RoboDK station: DemoFactorySimulation.rdk

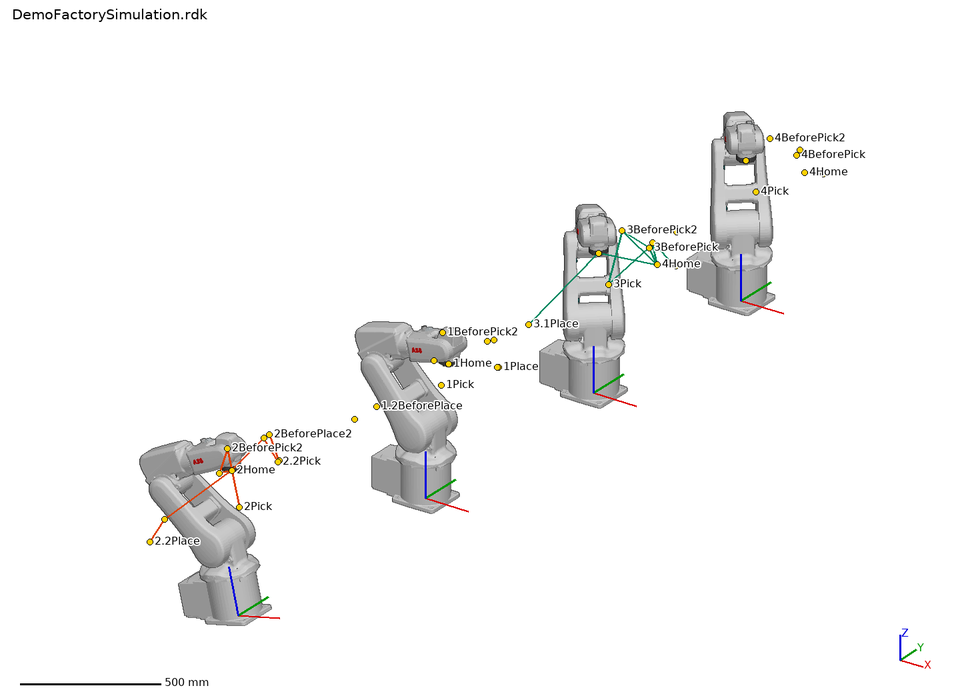
[picture v0: the station drawn from its stored meshes, robots at their saved joint values, targets as dots, program paths as lines]
Station RDTSDemoBasketLine. Poses are relative to the parent item; angles as X-Y-Z fixed-axis rotations.
Station parameters (name, value as stored): 1MoveToPick, 0, 1MakePick, 0, 1PickObjOK, 0, 1MoveToPlace, 0, 1MakePlace, 0, 1PlaceObjOK, 0, 1Waitting, 1, 2MoveToPick, 0, 2MakePick, 0, 2PickObjOK, 1, 2MoveToPlace, 0, 2MakePlace, 0, 2PlaceObjOK, 0, 2Waitting, 1, 3MoveToPick, 0, 3MakePick, 1, 3PickObjOK, 0, 3MoveToPlace, 0, 3MakePlace, 0, 3PlaceObjOK, 0, 3Waitting, 0, 4MoveToPick, 0, 4MakePick, 0, 4PickObjOK, 0, 4MoveToPlace, 0, 4MakePlace, 0, 4PlaceObjOK, 0, 4Waitting, 1, 5MoveToPick, 0, 5MakePick, 0, 5PickObjOK, 0, 5MoveToPlace, 0, 5MakePlace, 0, 5PlaceObjOK, 0, 5Waitting, 1
  - frame Robot1Base at (0, 605.93, 0) mm
    - robot Robot1 (model ABB IRB 120-3/0.6): 6 axes, payload 3 kg, reach 580 mm, repeatability 0.01 mm, weight 25 kg
        modified DH rows (alpha deg, a mm, theta deg, d mm): 0, 0, 0, 290; -90, 0, -90, 0; 0, 270, 0, 0; -90, 70, 0, 302; 90, 0, 0, 0; -90, 0, 180, 72
        joint limits [-165, -110, -90, -160, -120, -400] to [165, 110, 70, 160, 120, 400]; home [0, 0, 0, 0, 0, 0]; saved at [0, -40.936, 28.088, 0, 105.49, 0]
    - target 1Home (Cartesian target) at (98.64, 0, 557.45) mm, rotated rx 180 ry -2.64 rz 180 deg; joints [0, -40.936, 28.088, 0, 105.49, 0] of Robot1
    - target 1BeforePick (Cartesian target) at (1.46, 49.24, 523.75) mm, rotated rx -179.78 ry 0.01 rz -91.44 deg; joints [88.62, -55.08, 38.94, -0.23, 106.13, 0] of Robot1
    - target 1BeforePick2 (Cartesian target) at (-74.07, 211.85, 549) mm, rotated rx -179.78 ry 0 rz -89.11 deg; joints [109.338, -16.563, 16.145, -0.21, 90.487, 18.449] of Robot1
    - target 1Pick (Cartesian target) at (-133.52, 287.77, 294.7) mm, rotated rx -179.78 ry 0.01 rz -90.69 deg; joints [114.936, 14.64, 34.94, -0.312, 40.509, 25.866] of Robot1
    - target 1AfterPick (Cartesian target) at (-74.07, 211.85, 549) mm, rotated rx -179.78 ry 0 rz -89.11 deg; joints [109.338, -16.563, 16.145, -0.21, 90.487, 18.449] of Robot1
    - target 1AfterPick2 (Cartesian target) at (1.46, 49.24, 523.75) mm, rotated rx -179.78 ry 0.01 rz -91.44 deg; joints [88.62, -55.08, 38.94, -0.23, 106.13, 0] of Robot1
    - target 1BeforePlace (Cartesian target) at (237.81, 40.67, 670.65) mm, rotated rx 180 ry -2.64 rz -180 deg; joints [9.575, -1.266, -21.78, 0.487, 115.649, 9.776] of Robot1
    - target 1BeforePlace2 (Cartesian target) at (266.26, 40.67, 684.58) mm, rotated rx 180 ry -2.64 rz 180 deg; joints [8.58, 7.385, -34.207, 0.452, 119.433, 8.793] of Robot1
    - target 1Place (Cartesian target) at (293.03, 32.57, 586.26) mm, rotated rx 180 ry -2.64 rz -180 deg; joints [6.273, 0.868, -6.289, 0.291, 98.045, 6.307] of Robot1
    - target 1AfterPlace (Cartesian target) at (266.26, 40.67, 684.58) mm, rotated rx 180 ry -2.64 rz 180 deg; joints [8.58, 7.385, -34.207, 0.452, 119.433, 8.793] of Robot1
    - target 1AfterPlace2 (Cartesian target) at (237.81, 40.67, 670.65) mm, rotated rx 180 ry -2.64 rz 180 deg; joints [9.575, -1.266, -21.78, 0.487, 115.649, 9.776] of Robot1
    - target 1.2BeforePick (Cartesian target) at (237.81, 40.67, 670.65) mm, rotated rx -180 ry -2.64 rz -180 deg; joints [9.575, -1.266, -21.78, 0.487, 115.649, 9.776] of Robot1
    - target 1.2Pick (Cartesian target) at (287.41, 32.18, 584.86) mm, rotated rx -180 ry -2.64 rz -180 deg; joints [6.316, -0.426, -4.718, 0.293, 97.768, 6.349] of Robot1
    - target 1.2AfterPick (Cartesian target) at (237.81, 40.67, 670.65) mm, rotated rx -180 ry -2.64 rz -180 deg; joints [9.575, -1.266, -21.78, 0.487, 115.649, 9.776] of Robot1
    - target 1.2BeforePlace (Cartesian target) at (0, -302, 481.65) mm, rotated rx 180 ry 0 rz 90 deg; joints [-90, -1.686, 15.888, 0, 75.798, 0] of Robot1
    - target 1.2Place (Cartesian target) at (-151.28, -221.68, 357.52) mm, rotated rx 180 ry 0 rz 90 deg; joints [-124.31, -2.755, 40.632, 0, 52.123, -34.31] of Robot1
    - target 1.2AfterPlace (Cartesian target) at (0, -302, 481.65) mm, rotated rx 180 ry 0 rz 90 deg; joints [-90, -1.686, 15.888, 0, 75.798, 0] of Robot1
  - program RobotProg1 (59 instructions, listed below)
  - frame Robot2Base at (0, -551.31, 0) mm, rotated rx 0 ry -12.89 rz 0 deg
    - robot Robot2 (model ABB IRB 120-3/0.6): 6 axes, payload 3 kg, reach 580 mm, repeatability 0.01 mm, weight 25 kg
        modified DH rows (alpha deg, a mm, theta deg, d mm): 0, 0, 0, 290; -90, 0, -90, 0; 0, 270, 0, 0; -90, 70, 0, 302; 90, 0, 0, 0; -90, 0, 180, 72
        joint limits [-165, -110, -90, -160, -120, -400] to [165, 110, 70, 160, 120, 400]; home [0, 0, 0, 0, 0, 0]; saved at [0, -40.936, 28.088, 0, 105.49, 0]
    - target 2Home (Cartesian target) at (98.64, 0, 557.45) mm, rotated rx 180 ry -2.64 rz 180 deg; joints [0, -40.936, 28.088, 0, 105.49, 0] of Robot2
    - target 2BeforePick (Cartesian target) at (1.46, 49.24, 523.75) mm, rotated rx -179.78 ry 0.01 rz -91.44 deg; joints [88.62, -55.08, 38.94, -0.23, 106.13, 0] of Robot2
    - target 2BeforePick2 (Cartesian target) at (-74.07, 211.85, 549) mm, rotated rx -179.78 ry 0 rz -89.11 deg; joints [109.338, -16.563, 16.145, -0.21, 90.487, 18.449] of Robot2
    - target 2Pick (Cartesian target) at (-133.52, 287.77, 294.7) mm, rotated rx -179.78 ry 0.01 rz -91.91 deg; joints [114.936, 14.64, 34.94, -0.312, 40.509, 27.079] of Robot2
    - target 2AfterPick (Cartesian target) at (-74.07, 211.85, 549) mm, rotated rx -179.78 ry 0 rz -89.11 deg; joints [109.338, -16.563, 16.145, -0.21, 90.487, 18.449] of Robot2
    - target 2AfterPick2 (Cartesian target) at (1.46, 49.24, 523.75) mm, rotated rx -179.78 ry 0.01 rz -91.44 deg; joints [88.62, -55.08, 38.94, -0.23, 106.13, 0] of Robot2
    - target 2BeforePlace (Cartesian target) at (237.81, 40.67, 670.65) mm, rotated rx 180 ry -2.64 rz -180 deg; joints [9.575, -1.266, -21.78, 0.487, 115.649, 9.776] of Robot2
    - target 2BeforePlace2 (Cartesian target) at (266.26, 40.67, 684.58) mm, rotated rx 180 ry -2.64 rz 180 deg; joints [8.58, 7.385, -34.207, 0.452, 119.433, 8.793] of Robot2
    - target 2Place (Cartesian target) at (293.25, 32.57, 591.05) mm, rotated rx 180 ry -2.64 rz 180 deg; joints [6.268, 1.267, -7.631, 0.292, 98.989, 6.307] of Robot2
    - target 2AfterPlace (Cartesian target) at (266.26, 40.67, 684.58) mm, rotated rx 180 ry -2.64 rz 180 deg; joints [8.58, 7.385, -34.207, 0.452, 119.433, 8.793] of Robot2
    - target 2AfterPlace2 (Cartesian target) at (237.81, 40.67, 670.65) mm, rotated rx 180 ry -2.64 rz 180 deg; joints [9.575, -1.266, -21.78, 0.487, 115.649, 9.776] of Robot2
    - target 2.2BeforePick (Cartesian target) at (237.81, 40.67, 670.65) mm, rotated rx -180 ry -2.64 rz -180 deg; joints [9.575, -1.266, -21.78, 0.487, 115.649, 9.776] of Robot2
    - target 2.2Pick (Cartesian target) at (287.41, 32.18, 584.86) mm, rotated rx -180 ry -2.64 rz -180 deg; joints [6.316, -0.426, -4.718, 0.293, 97.768, 6.349] of Robot2
    - target 2.2AfterPick (Cartesian target) at (237.81, 40.67, 670.65) mm, rotated rx -180 ry -2.64 rz -180 deg; joints [9.575, -1.266, -21.78, 0.487, 115.649, 9.776] of Robot2
    - target 2.2BeforePlace (Cartesian target) at (0, -302, 481.65) mm, rotated rx 180 ry 0 rz 90 deg; joints [-90, -1.686, 15.888, 0, 75.798, 0] of Robot2
    - target 2.2Place (Cartesian target) at (-151.28, -221.68, 357.52) mm, rotated rx 180 ry 0 rz 90 deg; joints [-124.31, -2.755, 40.632, 0, 52.123, -34.31] of Robot2
    - target 2.2AfterPlace (Cartesian target) at (0, -302, 481.65) mm, rotated rx 180 ry 0 rz 90 deg; joints [-90, -1.686, 15.888, 0, 75.798, 0] of Robot2
  - program RobotProg2 (59 instructions, listed below)
  - frame Robot3Base at (0, 1644.74, 0) mm
    - robot Robot3 (model ABB IRB 120-3/0.6): 6 axes, payload 3 kg, reach 580 mm, repeatability 0.01 mm, weight 25 kg
        modified DH rows (alpha deg, a mm, theta deg, d mm): 0, 0, 0, 290; -90, 0, -90, 0; 0, 270, 0, 0; -90, 70, 0, 302; 90, 0, 0, 0; -90, 0, 180, 72
        joint limits [-165, -110, -90, -160, -120, -400] to [165, 110, 70, 160, 120, 400]; home [0, 0, 0, 0, 0, 0]; saved at [-48.899, -24.574, 6.021, 0.542, 108.231, 40.826]
    - target 4Home (Cartesian target) at (262.7, 17.2, 573.39) mm, rotated rx 179.91 ry 0.6 rz -179.52 deg; joints [3.731, -7.418, 4.046, 0.057, 92.769, 3.257] of Robot3
    - target 3BeforePick (Cartesian target) at (168.05, 102.25, 580.49) mm, rotated rx 175.96 ry 3.61 rz -144.21 deg; joints [29.71, -21.07, 13.293, 4.417, 94.607, -5.734] of Robot3
    - target 3BeforePick2 (Cartesian target) at (16.7, 152.98, 583.81) mm, rotated rx -179.66 ry 5.4 rz -92.3 deg; joints [83.754, -29.723, 17.773, 0.036, 96.534, -3.924] of Robot3
    - target 3Pick (Cartesian target) at (-130.61, 278.87, 281.48) mm, rotated rx -179.66 ry 5.4 rz -92.3 deg; joints [115.76, 13.813, 39.181, -5.284, 32.502, 32.421] of Robot3
    - target 3Place (Cartesian target) at (339.21, 24.19, 586.4) mm, rotated rx 179.91 ry 0.6 rz -179.52 deg; joints [4.067, 9.967, -16.219, 0.054, 95.647, 3.595] of Robot3
    - target 3BeforePlace (Cartesian target) at (240.47, 19.38, 654.16) mm, rotated rx 179.91 ry 0.6 rz -179.52 deg; joints [4.594, -4.403, -15.131, 0.051, 108.929, 4.134] of Robot3
    - target 3.1Place (Cartesian target) at (-136.77, -205.36, 314.46) mm, rotated rx 179.4 ry -0.09 rz 90.45 deg; joints [-123.793, -2.069, 49.122, 0.647, 43.362, -34.71] of Robot3
    - target 3.1BeforePlace (Cartesian target) at (100.51, -114.23, 626) mm, rotated rx 179.4 ry -0.09 rz 90.45 deg; joints [-48.899, -24.574, 6.021, 0.542, 108.231, 40.826] of Robot3
  - program RobotProg3 (59 instructions, listed below)
  - frame RobotBase4 at (0, 2557.3, 0) mm
    - robot Robot4 (model ABB IRB 120-3/0.6): 6 axes, payload 3 kg, reach 580 mm, repeatability 0.01 mm, weight 25 kg
        modified DH rows (alpha deg, a mm, theta deg, d mm): 0, 0, 0, 290; -90, 0, -90, 0; 0, 270, 0, 0; -90, 70, 0, 302; 90, 0, 0, 0; -90, 0, 180, 72
        joint limits [-165, -110, -90, -160, -120, -400] to [165, 110, 70, 160, 120, 400]; home [0, 0, 0, 0, 0, 0]; saved at [-48.899, -24.574, 6.021, 0.542, 108.231, 40.826]
    - target 4Home (Cartesian target) at (262.7, 17.2, 573.39) mm, rotated rx 179.91 ry 0.6 rz -179.52 deg; joints [3.731, -7.418, 4.046, 0.057, 92.769, 3.257] of Robot4
    - target 4BeforePick (Cartesian target) at (168.05, 102.25, 580.49) mm, rotated rx 175.96 ry 3.61 rz -144.21 deg; joints [29.71, -21.07, 13.293, 4.417, 94.607, -5.734] of Robot4
    - target 4BeforePick2 (Cartesian target) at (16.7, 152.98, 583.81) mm, rotated rx -179.66 ry 5.4 rz -92.3 deg; joints [83.754, -29.723, 17.773, 0.036, 96.534, -3.924] of Robot4
    - target 4Pick (Cartesian target) at (-130.61, 278.87, 281.48) mm, rotated rx -179.66 ry 5.4 rz -92.3 deg; joints [115.76, 13.813, 39.181, -5.284, 32.502, 32.421] of Robot4
    - target 4Place (Cartesian target) at (339.21, 24.19, 586.4) mm, rotated rx 179.91 ry 0.6 rz -179.52 deg; joints [4.067, 9.967, -16.219, 0.054, 95.647, 3.595] of Robot4
    - target 4BeforePlace (Cartesian target) at (240.47, 19.38, 654.16) mm, rotated rx 179.91 ry 0.6 rz -179.52 deg; joints [4.594, -4.403, -15.131, 0.051, 108.929, 4.134] of Robot4
    - target 4.1Place (Cartesian target) at (-136.77, -205.36, 314.46) mm, rotated rx 179.4 ry -0.09 rz 90.45 deg; joints [-123.793, -2.069, 49.122, 0.647, 43.362, -34.71] of Robot4
    - target 4.1BeforePlace (Cartesian target) at (100.51, -114.23, 626) mm, rotated rx 179.4 ry -0.09 rz 90.45 deg; joints [-48.899, -24.574, 6.021, 0.542, 108.231, 40.826] of Robot4
  - program RobotProg3 (59 instructions, listed below)
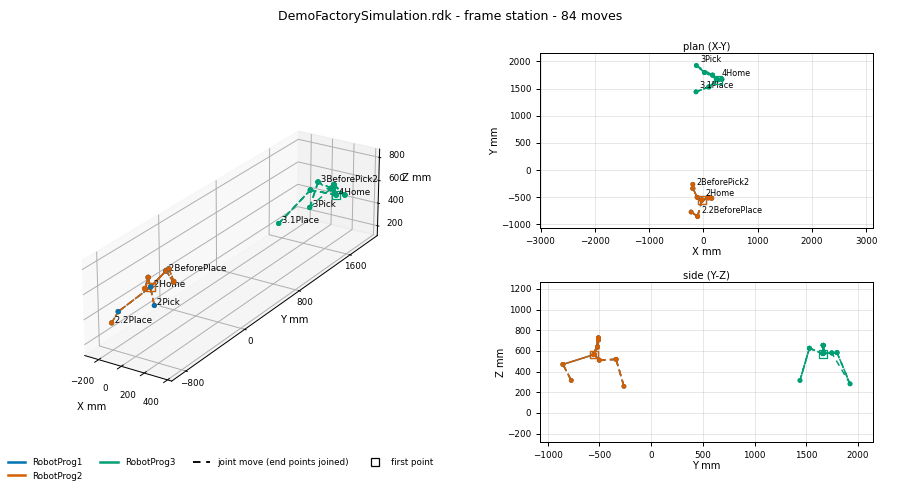
[picture p0: tool path of DemoFactorySimulation.rdk in frame station, 84 of 84 moves have a stored position in this frame; points joined in program order, loops and branches not executed]

--- program RobotProg1 (robot Robot1) ---
  Set Ref.: Robot1Base
  MoveJ (2Home)
  Set 1MakePick=0
  Set 1PickObjOK=0
  Set 1MakePlace=0
  Set 1PlaceObjOK=0
  Wait 1MoveToPick=1
  Set 1Waitting=0
  MoveJ (2BeforePick)
  MoveJ (2BeforePick2)
  MoveJ (2Pick)
  Set 1MakePick=1
  Wait 1PickObjOK=1
  Set 1MakePick=0
  暂停 2.0 s
  MoveJ (2AfterPick)
  MoveJ (2AfterPick2)
  MoveJ (2Home)
  Set 1Waitting=1
  Wait 1MoveToPlace=1
  Set 1Waitting=0
  MoveJ (2BeforePlace)
  MoveJ (2BeforePlace2)
  MoveJ (2Place)
  Set 1MakePlace=1
  Wait 1PlaceObjOK=1
  Set 1MakePlace=0
  暂停 1.0 s
  MoveJ (2AfterPlace)
  MoveJ (2AfterPlace2)
  MoveJ (2Home)
  Set 1Waitting=1
  暂停 2.5 s
  Set 1MakePick=0
  Set 1PickObjOK=0
  Set 1MakePlace=0
  Set 1PlaceObjOK=0
  Wait 1MoveToPick=1
  Set 1Waitting=0
  MoveJ (2.2BeforePick)
  MoveJ (2.2Pick)
  Set 1MakePick=1
  Wait 1PickObjOK=1
  Set 1MakePick=0
  暂停 2.0 s
  MoveJ (2.2AfterPick)
  MoveJ (2Home)
  Set 1Waitting=1
  Wait 1MoveToPlace=1
  Set 1Waitting=0
  MoveJ (2.2BeforePlace)
  MoveJ (2.2Place)
  Set 1MakePlace=1
  Wait 1PlaceObjOK=1
  Set 1MakePlace=0
  暂停 1.0 s
  MoveJ (2.2AfterPlace)
  MoveJ (2Home)
  Set 1Waitting=1

--- program RobotProg2 (robot Robot2) ---
  设置参考: Robot2Base
  MoveJ (2Home)
  Set 2MakePick=0
  Set 2PickObjOK=0
  Set 2MakePlace=0
  Set 2PlaceObjOK=0
  Wait 2MoveToPick=1
  Set 2Waitting=0
  MoveJ (2BeforePick)
  MoveJ (2BeforePick2)
  MoveJ (2Pick)
  Set 2MakePick=1
  Wait 2PickObjOK=1
  Set 2MakePick=0
  暂停 2.0 s
  MoveJ (2AfterPick)
  MoveJ (2AfterPick2)
  MoveJ (2Home)
  Set 2Waitting=1
  Wait 2MoveToPlace=1
  Set 2Waitting=0
  MoveJ (2BeforePlace)
  MoveJ (2BeforePlace2)
  MoveJ (2Place)
  Set 2MakePlace=1
  Wait 2PlaceObjOK=1
  Set 2MakePlace=0
  暂停 1.0 s
  MoveJ (2AfterPlace)
  MoveJ (2AfterPlace2)
  MoveJ (2Home)
  Set 2Waitting=1
  暂停 2.5 s
  Set 2MakePick=0
  Set 2PickObjOK=0
  Set 2MakePlace=0
  Set 2PlaceObjOK=0
  Wait 2MoveToPick=1
  Set 2Waitting=0
  MoveJ (2.2BeforePick)
  MoveJ (2.2Pick)
  Set 2MakePick=1
  Wait 2PickObjOK=1
  Set 2MakePick=0
  暂停 2.0 s
  MoveJ (2.2AfterPick)
  MoveJ (2Home)
  Set 2Waitting=1
  Wait 2MoveToPlace=1
  Set 2Waitting=0
  MoveJ (2.2BeforePlace)
  MoveJ (2.2Place)
  Set 2MakePlace=1
  Wait 2PlaceObjOK=1
  Set 2MakePlace=0
  暂停 1.0 s
  MoveJ (2.2AfterPlace)
  MoveJ (2Home)
  Set 2Waitting=1

--- program RobotProg3 (robot Robot3) ---
  Set Ref.: Robot3Base
  MoveJ (3Home) -> target 4Home
  Set 3MakePick=0
  Set 3PickObjOK=0
  Set 3MakePlace=0
  Set 3PlaceObjOK=0
  Wait 3MoveToPick=1
  Set 3Waitting=0
  MoveJ (3BeforePick)
  MoveJ (3BeforePick2)
  MoveJ (3Pick)
  Set 3MakePick=1
  Wait 3PickObjOK=1
  Set 3MakePick=0
  暂停 2.0 s
  MoveJ (3BeforePick) -> target 3BeforePick2
  MoveJ (3BeforePick) -> target 3BeforePick2
  MoveJ (3Home) -> target 4Home
  Set 3Waitting=1
  Wait 3MoveToPlace=1
  Set 3Waitting=0
  MoveJ (3BeforePlace)
  MoveJ (3BeforePlace)
  MoveJ (3Place)
  Set 3MakePlace=1
  Wait 3PlaceObjOK=1
  Set 3MakePlace=0
  暂停 1.0 s
  MoveJ (3BeforePlace)
  MoveJ (3BeforePlace)
  MoveJ (3Home) -> target 4Home
  Set 3Waitting=1
  暂停 2.5 s
  Set 3MakePick=0
  Set 3PickObjOK=0
  Set 3MakePlace=0
  Set 3PlaceObjOK=0
  Wait 3MoveToPick=1
  Set 3Waitting=0
  MoveJ (3BeforePlace)
  MoveJ (3Place)
  Set 3MakePick=1
  Wait 3PickObjOK=1
  Set 3MakePick=0
  暂停 2.0 s
  MoveJ (3BeforePlace)
  MoveJ (3Home) -> target 4Home
  Set 3Waitting=1
  Wait 3MoveToPlace=1
  Set 3Waitting=0
  MoveJ (3.1BeforePlace)
  MoveJ (3.1Place)
  Set 3MakePlace=1
  Wait 3PlaceObjOK=1
  Set 3MakePlace=0
  暂停 1.0 s
  MoveJ (3.1BeforePlace)
  MoveJ (3Home) -> target 4Home
  Set 3Waitting=1

--- program RobotProg3 (robot Robot4) ---
  Set Ref.: RobotBase4
  MoveJ (4Home)
  Set 4MakePick=0
  Set 4PickObjOK=0
  Set 4MakePlace=0
  Set 4PlaceObjOK=0
  Wait 4MoveToPick=1
  Set 4Waitting=0
  MoveJ (4BeforePick) -> target 3BeforePick
  MoveJ (4BeforePick2) -> target 3BeforePick2
  MoveJ (4Pick) -> target 3Pick
  Set 4MakePick=1
  Wait 4PickObjOK=1
  Set 4MakePick=0
  暂停 2.0 s
  MoveJ (3BeforePick)
  MoveJ (3BeforePick)
  MoveJ (4Home)
  Set 4Waitting=1
  Wait 4MoveToPlace=1
  Set 4Waitting=0
  MoveJ (3BeforePlace)
  MoveJ (3BeforePlace)
  MoveJ (3Place)
  Set 4MakePlace=1
  Wait 4PlaceObjOK=1
  Set 4MakePlace=0
  暂停 1.0 s
  MoveJ (3BeforePlace)
  MoveJ (3BeforePlace)
  MoveJ (4Home)
  Set 4Waitting=1
  暂停 2.5 s
  Set 4MakePick=0
  Set 4PickObjOK=0
  Set 4MakePlace=0
  Set 4PlaceObjOK=0
  Wait 4MoveToPick=1
  Set 4Waitting=0
  MoveJ (3BeforePlace)
  MoveJ (3Place)
  Set 4MakePick=1
  Wait 4PickObjOK=1
  Set 4MakePick=0
  暂停 2.0 s
  MoveJ (3BeforePlace)
  MoveJ (4Home)
  Set 4Waitting=1
  Wait 4MoveToPlace=1
  Set 4Waitting=0
  MoveJ (3.1BeforePlace)
  MoveJ (3.1Place)
  Set 4MakePlace=1
  Wait 4PlaceObjOK=1
  Set 4MakePlace=0
  暂停 1.0 s
  MoveJ (3.1BeforePlace)
  MoveJ (4Home)
  Set 4Waitting=1
